INTERFACE ITF_MCHMIPrepareScreen_05_XX_Init

METHOD PUBLIC LinkDataHMI_05_XX : BOOL
VAR_INPUT
	refstData				: REFERENCE TO ST_MCHMIPrepareScreen_05_XX;
END_VAR
END_METHOD

END_INTERFACE

(* stored: Version 1.1.0.1
   Itf ITF_MCHMIPrepareScreen_05_XX_Init: Id {4fbbd5eb-0e76-055c-1448-52866d302f03}
   Method LinkDataHMI_05_XX: Id {48c4ef85-822d-075e-1c60-145b4256a086} *)
